FUNCTION F_HasContext : BOOL
VAR_INPUT
	nContext: DWORD;
	nSearchContext: DWORD;
END_VAR
VAR
END_VAR


F_HasContext:= (nContext > 0) AND (((nContext AND nSearchContext) > 0) OR (nSearchContext = E_DataSourceContext.eContext_Unknown));

END_FUNCTION

(* stored: POU F_HasContext: Id 8797fec5-2773-443c-a342-57136dda5ce3, SpecialFunc None *)
